FUNCTION CONTROLWORD_STATE_CHANGE : WORD
VAR_INPUT
	Current_State 		: E_Statemachine_State;
	Target_State 		: E_Statemachine_State;	
END_VAR
VAR
	Controlword 		: WORD;
END_VAR

CASE Current_State OF
    E_Statemachine_State.Not_ready_to_switch_on:		// Wait for 'Switch on disabled'
		Controlword := E_Statemachine_Transition_Controlword.Switch_on_disabled;

	E_Statemachine_State.Switch_on_disabled:
		CASE Target_State OF
			E_Statemachine_State.Ready_to_switch_on:	Controlword := E_Statemachine_Transition_Controlword.Ready_to_switch_on;				
			E_Statemachine_State.Switched_on:			Controlword := E_Statemachine_Transition_Controlword.Ready_to_switch_on;				
			E_Statemachine_State.Operation_enabled:		Controlword := E_Statemachine_Transition_Controlword.Ready_to_switch_on;				
		ELSE
			Controlword := E_Statemachine_Transition_Controlword.Switch_on_disabled;			
		END_CASE

	E_Statemachine_State.Ready_to_switch_on:
		CASE Target_State OF
			E_Statemachine_State.Switch_on_disabled:	Controlword := E_Statemachine_Transition_Controlword.Switch_on_disabled;			
			E_Statemachine_State.Switched_on:			Controlword := E_Statemachine_Transition_Controlword.Switched_on;			
			E_Statemachine_State.Operation_enabled:		Controlword := E_Statemachine_Transition_Controlword.Switched_on;					
		ELSE
			Controlword := E_Statemachine_Transition_Controlword.Ready_to_switch_on;			
		END_CASE
				
	E_Statemachine_State.Switched_on:
		CASE Target_State OF
			E_Statemachine_State.Switch_on_disabled:	Controlword := E_Statemachine_Transition_Controlword.Switch_on_disabled;		
			E_Statemachine_State.Ready_to_switch_on:	Controlword := E_Statemachine_Transition_Controlword.Ready_to_switch_on;	
			E_Statemachine_State.Operation_enabled:		Controlword := E_Statemachine_Transition_Controlword.Operation_enabled;				
		ELSE
			CONTROLWORD_STATE_CHANGE := E_Statemachine_Transition_Controlword.Switched_on;				
		END_CASE
		
	E_Statemachine_State.Operation_enabled:
		CASE Target_State OF
			E_Statemachine_State.Switch_on_disabled:	Controlword := E_Statemachine_Transition_Controlword.Switch_on_disabled;		
			E_Statemachine_State.Ready_to_switch_on:	Controlword := E_Statemachine_Transition_Controlword.Ready_to_switch_on;	
			E_Statemachine_State.Switched_on:			Controlword := E_Statemachine_Transition_Controlword.Switched_on;		
			E_Statemachine_State.Quick_stop_active:		Controlword := E_Statemachine_Transition_Controlword.Quick_stop_active;				
		ELSE
			Controlword := E_Statemachine_Transition_Controlword.Operation_enabled;	;			
		END_CASE
		
	E_Statemachine_State.Quick_stop_active:				
		CASE Target_State OF
			E_Statemachine_State.Switch_on_disabled:	Controlword := E_Statemachine_Transition_Controlword.Switch_on_disabled;		
			E_Statemachine_State.Ready_to_switch_on:	Controlword := E_Statemachine_Transition_Controlword.Switch_on_disabled;	
			E_Statemachine_State.Switched_on:			Controlword := E_Statemachine_Transition_Controlword.Switch_on_disabled;	
			E_Statemachine_State.Operation_enabled:		Controlword := E_Statemachine_Transition_Controlword.Switch_on_disabled;	// Not recommennded to support to switch back directly			
		ELSE
			Controlword := 16#2;			
		END_CASE
		
	E_Statemachine_State.Fault_reaction_active:			// Wait for 'Fault'
		Controlword := E_Statemachine_Transition_Controlword.Switch_on_disabled;
		
	E_Statemachine_State.Fault:
		CASE Target_State OF
 			E_Statemachine_State.Switch_on_disabled, E_Statemachine_State.Ready_to_switch_on, E_Statemachine_State.Switched_on, E_Statemachine_State.Operation_enabled:
				// Toggle the Fault reset bit
				IF PDO.Controlword = E_Statemachine_Transition_Controlword.Faultreset_step_2 THEN	Controlword := E_Statemachine_Transition_Controlword.Faultreset_step_1; ELSE Controlword := E_Statemachine_Transition_Controlword.Faultreset_step_2; END_IF
		ELSE
			Controlword := E_Statemachine_Transition_Controlword.Switch_on_disabled;
		END_CASE;
	
ELSE
    Controlword := 16#0;
	
END_CASE;

// Return the new controlword
CONTROLWORD_STATE_CHANGE := Controlword;

END_FUNCTION

(* stored: Version 1.1.0.1, ProductVersion 3.1.4024.12
   POU CONTROLWORD_STATE_CHANGE: Id {e061c73d-e1b6-4378-816e-f68084458999}, SpecialFunc None *)
